{attribute 'qualified_only'}
VAR_GLOBAL
	Section : ARRAY [1..4] OF ST_Section_Base;
END_VAR

(* stored: Version 1.1.0.1, ProductVersion 3.1.4024.11
   GVL LCP: Id {99f22dc7-bbc0-423c-a5af-e55fc8eb108e} *)
